{attribute 'no_explicit_call' := 'do not call this FB directly'}{attribute 'enable_dynamic_creation'}
FUNCTION_BLOCK OutputPort EXTENDS Disposable IMPLEMENTS I_OutputPort
VAR
	_name : T_MAXSTRING;
	_dataType : T_MAXSTRING;
	data : Data;
	eventEmitter : EventEmitter;
END_VAR

METHOD PUBLIC Accept
VAR_INPUT
	Visitor : I_OutputPortVisitor;
END_VAR
Visitor.VisitOutputPort(this^);
END_METHOD

PROPERTY PUBLIC Data : T_MAXSTRING
GET
OutputPort.Data := _dataType;
END_GET
END_PROPERTY

METHOD PRIVATE EmitOnOutputPortChangeEvent
VAR_INPUT
	PortChanged : I_OutputPort;
END_VAR
VAR
	pOutputPortChangeEvent : POINTER TO OutputPortChangedEvent;
END_VAR
pOutputPortChangeEvent := __NEW(OutputPortChangedEvent(TargetOutputPort := PortChanged));
eventEmitter.Emit('OnOutputPortChanged',pOutputPortChangeEvent^);
pOutputPortChangeEvent^.Dispose();
END_METHOD

METHOD FB_init : BOOL
VAR_INPUT
	bInitRetains : BOOL; // if TRUE, the retain variables are initialized (warm start / cold start)
	bInCopyCode : BOOL;  // if TRUE, the instance afterwards gets moved into the copy code (online change)
	Name : T_MAXSTRING;
	DataType : T_MAXSTRING;
	Parent : I_HaveOutputPorts;
END_VAR
_name := Name;
_dataType := DataType;

IF Parent = 0 THEN
	RETURN;
END_IF

Parent.AddOutputPort(THIS^);
END_METHOD

PROPERTY PUBLIC Name : T_MAXSTRING
GET
Name := _name;
END_GET
END_PROPERTY

METHOD PUBLIC OffEvent
VAR_INPUT
	EventName : T_MaxString;
	EventHandler : I_EventHandler;
END_VAR
eventEmitter.OffEvent(EventName, EventHandler);
END_METHOD

METHOD PUBLIC OnceEvent
VAR_INPUT
	EventName : T_MaxString;
	EventHandler : I_EventHandler;
END_VAR
eventEmitter.OnceEvent(EventName, EventHandler);
END_METHOD

METHOD PUBLIC OnEvent
VAR_INPUT
	EventName : T_MaxString;
	EventHandler : I_EventHandler;
END_VAR
eventEmitter.OnEvent(EventName, EventHandler);
END_METHOD

METHOD PUBLIC TryGet : BOOL;
VAR_INPUT
	Value : ANY;
END_VAR
TryGet := OutputPort.Data.TryGet(Value);
END_METHOD

METHOD PUBLIC TryGetTo : BOOL;
VAR_INPUT
	Destination : PVOID;
	DestinationSize : UDINT;
END_VAR
TryGetTo := OutputPort.Data.TryGetTo(Destination, DestinationSize);
END_METHOD

METHOD PUBLIC TrySet : BOOL;
VAR_INPUT
	Value : ANY;
END_VAR
TrySet := OutputPort.Data.TrySet(Value);
END_METHOD

METHOD PUBLIC TrySetFrom : BOOL;
VAR_INPUT
	SourceAddress : PVOID;
	SourceSize : UDINT;
END_VAR
IF NOT OutputPort.Data.TrySetFrom(SourceAddress, SourceSize) THEN
	RETURN;
END_IF

EmitOnOutputPortChangeEvent(THIS^);
TrySetFrom := TRUE;
END_METHOD

END_FUNCTION_BLOCK

(* stored: Version 1.1.0.1, ProductVersion 3.1.4024.12
   POU OutputPort: Id {4c7e0bce-9eb0-0f6a-044f-6a3cfc8b783d}, SpecialFunc None
   Folder Constructor: Id {677256cd-e8af-081b-2804-5689f5f4149b}
   Folder Private: Id {6f5f4b13-ef19-01e5-075e-0ea3b801d3d7}
   Method Accept: Id {685a8b40-a5b2-0491-3a06-acbf37dad5a1}
   Property Data: Id {eb163034-b0fd-0fe3-0fa5-fd0220399dfb}
   Get Get: Id {7534416c-ca26-06ef-2b8b-0ad13dd0d8f6}
   Method EmitOnOutputPortChangeEvent: Id {4cedd9f2-3d84-035e-18ce-b7ebc3af2524}
   Method FB_init: Id {1ba1d2d7-341d-0e8e-05ef-f5346255db4e}
   Property Name: Id {a6251d93-37b5-06d7-00eb-bc1261f23075}
   Get Get: Id {66530c4b-9811-0535-0d83-3db73e2195f3}
   Method OffEvent: Id {5f0c98a6-efae-06ce-0d53-00d24017a360}
   Method OnceEvent: Id {33aa55e6-cc64-0804-1f68-fe127e9ffd59}
   Method OnEvent: Id {83584882-e2df-000f-0211-5ef5ee02b990}
   Method TryGet: Id {d7f053a1-edb3-045f-2e85-d7d160cdb265}
   Method TryGetTo: Id {6e5c850e-5dc7-0ca4-0094-d63313848019}
   Method TrySet: Id {1e1c2da9-f2e1-0401-2df7-d89f92cc9a3e}
   Method TrySetFrom: Id {76d02626-79e8-0585-25de-a6810fcf20bc} *)
